// TIA Portal V20 export
TYPE "Stroke"
   STRUCT
      LinaAxis : Struct
         X : "MaxMin";
         Y : "MaxMin";
         Z { S7_SetPoint := 'True'} : "MaxMin";
      END_STRUCT;
      AngAxis : Struct
         "B" : "MaxMin";
         C : "MaxMin";
      END_STRUCT;
   END_STRUCT;
END_TYPE
